INTERFACE InterfaceFuture

PROPERTY active_futures : UINT
GET
END_GET
END_PROPERTY

METHOD execute : BOOL
VAR_INPUT
END_VAR
END_METHOD

METHOD init : BOOL
VAR_INPUT
END_VAR
END_METHOD

METHOD quit : BOOL
VAR_INPUT
END_VAR
END_METHOD

PROPERTY result : HRESULT
GET
END_GET
END_PROPERTY

END_INTERFACE

(* stored: Version 1.1.0.1, ProductVersion 3.1.4024.12
   Itf InterfaceFuture: Id {882bc581-e126-40c6-885e-c12ccc2f0bb9}
   Property active_futures: Id {2d416ece-2dc1-4b01-a1fe-d0b196d80eaa}
   Get Get: Id {9f74c5c8-3fa8-4c0a-9b16-6bb5d20b0f71}
   Method execute: Id {4a0b4721-18ea-4776-928a-5b24c49dda75}
   Method init: Id {d56cdce8-543b-417d-80a1-0c782146e5ce}
   Method quit: Id {12e3433d-9567-4756-bdca-54fc6f4c2614}
   Property result: Id {091e3808-1f21-4039-8bcc-e07988c843df}
   Get Get: Id {3dfc56f5-414c-4e9f-8318-d6a9044e8070} *)
